(* PLC project booster_compressor, TwinForge TwinForge 0.1.0 *)
(* stored: creationDateTime 2026-07-23T22:04:36.214256+00:00 *)

PROGRAM MainProgram
  VAR
    TF_Cmp_MainProgram_R00_AnalogAlarms_0_1 : BOOL;  (* TwinForge comparison result for R00_AnalogAlarms rung 0 *)
    TF_Cmp_MainProgram_R00_AnalogAlarms_1_1 : BOOL;  (* TwinForge comparison result for R00_AnalogAlarms rung 1 *)
    TF_Cmp_MainProgram_R00_AnalogAlarms_2_1 : BOOL;  (* TwinForge comparison result for R00_AnalogAlarms rung 2 *)
    TF_Cmp_MainProgram_R00_AnalogAlarms_3_1 : BOOL;  (* TwinForge comparison result for R00_AnalogAlarms rung 3 *)
    TF_Cmp_MainProgram_R00_AnalogAlarms_4_1 : BOOL;  (* TwinForge comparison result for R00_AnalogAlarms rung 4 *)
    TF_Cmp_MainProgram_R00_AnalogAlarms_5_1 : BOOL;  (* TwinForge comparison result for R00_AnalogAlarms rung 5 *)
    TF_Cmp_MainProgram_R03_Trips_5_1 : BOOL;  (* TwinForge comparison result for R03_Trips rung 5 *)
    TF_Cmp_MainProgram_R03_Trips_7_1 : BOOL;  (* TwinForge comparison result for R03_Trips rung 7 *)
    TF_Cmp_MainProgram_R03_Trips_9_1 : BOOL;  (* TwinForge comparison result for R03_Trips rung 9 *)
    TF_Cmp_MainProgram_R03_Trips_10_1 : BOOL;  (* TwinForge comparison result for R03_Trips rung 10 *)
    TF_Cmp_MainProgram_R03_Trips_14_1 : BOOL;  (* TwinForge comparison result for R03_Trips rung 14 *)
    TF_Cmp_MainProgram_R03_Trips_15_1 : BOOL;  (* TwinForge comparison result for R03_Trips rung 15 *)
    TF_Cmp_MainProgram_R03_Trips_16_1 : BOOL;  (* TwinForge comparison result for R03_Trips rung 16 *)
    TF_Cmp_MainProgram_R03_Trips_17_1 : BOOL;  (* TwinForge comparison result for R03_Trips rung 17 *)
    TF_Cmp_MainProgram_R03_Trips_18_1 : BOOL;  (* TwinForge comparison result for R03_Trips rung 18 *)
    TF_Cmp_MainProgram_R03_Trips_19_1 : BOOL;  (* TwinForge comparison result for R03_Trips rung 19 *)
    TF_Cmp_MainProgram_R03_Trips_20_1 : BOOL;  (* TwinForge comparison result for R03_Trips rung 20 *)
    TF_Cmp_MainProgram_R03_Trips_21_1 : BOOL;  (* TwinForge comparison result for R03_Trips rung 21 *)
    TF_Cmp_MainProgram_R03_Trips_22_1 : BOOL;  (* TwinForge comparison result for R03_Trips rung 22 *)
    TF_Cmp_MainProgram_R04_Sequence_5_1 : BOOL;  (* TwinForge comparison result for R04_Sequence rung 5 *)
    TF_Cmp_MainProgram_R04_Sequence_5_2 : BOOL;  (* TwinForge comparison result for R04_Sequence rung 5 *)
    TF_Cmp_MainProgram_R04_Sequence_5_3 : BOOL;  (* TwinForge comparison result for R04_Sequence rung 5 *)
    TF_Cmp_MainProgram_R04_Sequence_6_1 : BOOL;  (* TwinForge comparison result for R04_Sequence rung 6 *)
    TF_Cmp_MainProgram_R04_Sequence_7_1 : BOOL;  (* TwinForge comparison result for R04_Sequence rung 7 *)
    TF_Cmp_MainProgram_R04_Sequence_8_1 : BOOL;  (* TwinForge comparison result for R04_Sequence rung 8 *)
    TF_Cmp_MainProgram_R04_Sequence_9_1 : BOOL;  (* TwinForge comparison result for R04_Sequence rung 9 *)
    TF_Cmp_MainProgram_R04_Sequence_9_2 : BOOL;  (* TwinForge comparison result for R04_Sequence rung 9 *)
    TF_Cmp_MainProgram_R04_Sequence_10_1 : BOOL;  (* TwinForge comparison result for R04_Sequence rung 10 *)
    TF_Cmp_MainProgram_R04_Sequence_10_2 : BOOL;  (* TwinForge comparison result for R04_Sequence rung 10 *)
    TF_Cmp_MainProgram_R04_Sequence_11_1 : BOOL;  (* TwinForge comparison result for R04_Sequence rung 11 *)
    TF_Cmp_MainProgram_R04_Sequence_11_2 : BOOL;  (* TwinForge comparison result for R04_Sequence rung 11 *)
    TF_Cmp_MainProgram_R04_Sequence_12_1 : BOOL;  (* TwinForge comparison result for R04_Sequence rung 12 *)
    TF_Cmp_MainProgram_R04_Sequence_13_1 : BOOL;  (* TwinForge comparison result for R04_Sequence rung 13 *)
    TF_Cmp_MainProgram_R04_Sequence_14_1 : BOOL;  (* TwinForge comparison result for R04_Sequence rung 14 *)
    TF_Cmp_MainProgram_R04_Sequence_15_1 : BOOL;  (* TwinForge comparison result for R04_Sequence rung 15 *)
    TF_Cmp_MainProgram_R04_Sequence_16_1 : BOOL;  (* TwinForge comparison result for R04_Sequence rung 16 *)
    TF_Cmp_MainProgram_R04_Sequence_17_1 : BOOL;  (* TwinForge comparison result for R04_Sequence rung 17 *)
    TF_Cmp_MainProgram_R04_Sequence_17_2 : BOOL;  (* TwinForge comparison result for R04_Sequence rung 17 *)
    TF_Cmp_MainProgram_R04_Sequence_18_1 : BOOL;  (* TwinForge comparison result for R04_Sequence rung 18 *)
    TF_Cmp_MainProgram_R04_Sequence_19_1 : BOOL;  (* TwinForge comparison result for R04_Sequence rung 19 *)
    TF_Cmp_MainProgram_R04_Sequence_20_1 : BOOL;  (* TwinForge comparison result for R04_Sequence rung 20 *)
    TF_Cmp_MainProgram_R04_Sequence_21_1 : BOOL;  (* TwinForge comparison result for R04_Sequence rung 21 *)
    TF_Cmp_MainProgram_R04_Sequence_22_1 : BOOL;  (* TwinForge comparison result for R04_Sequence rung 22 *)
    TF_Cmp_MainProgram_R04_Sequence_22_2 : BOOL;  (* TwinForge comparison result for R04_Sequence rung 22 *)
    TF_Cmp_MainProgram_R04_Sequence_23_1 : BOOL;  (* TwinForge comparison result for R04_Sequence rung 23 *)
    TF_Cmp_MainProgram_R04_Sequence_24_1 : BOOL;  (* TwinForge comparison result for R04_Sequence rung 24 *)
    TF_Cmp_MainProgram_R04_Sequence_25_1 : BOOL;  (* TwinForge comparison result for R04_Sequence rung 25 *)
    TF_Cmp_MainProgram_R04_Sequence_26_1 : BOOL;  (* TwinForge comparison result for R04_Sequence rung 26 *)
    TF_Cmp_MainProgram_R04_Sequence_26_2 : BOOL;  (* TwinForge comparison result for R04_Sequence rung 26 *)
    TF_Cmp_MainProgram_R04_Sequence_27_1 : BOOL;  (* TwinForge comparison result for R04_Sequence rung 27 *)
    TF_Cmp_MainProgram_R04_Sequence_28_1 : BOOL;  (* TwinForge comparison result for R04_Sequence rung 28 *)
    TF_Cmp_MainProgram_R04_Sequence_29_1 : BOOL;  (* TwinForge comparison result for R04_Sequence rung 29 *)
    TF_Cmp_MainProgram_R04_Sequence_30_1 : BOOL;  (* TwinForge comparison result for R04_Sequence rung 30 *)
    TF_Cmp_MainProgram_R04_Sequence_31_1 : BOOL;  (* TwinForge comparison result for R04_Sequence rung 31 *)
    TF_Cmp_MainProgram_R04_Sequence_32_1 : BOOL;  (* TwinForge comparison result for R04_Sequence rung 32 *)
    TF_Cmp_MainProgram_R04_Sequence_33_1 : BOOL;  (* TwinForge comparison result for R04_Sequence rung 33 *)
    TF_Cmp_MainProgram_R04_Sequence_33_2 : BOOL;  (* TwinForge comparison result for R04_Sequence rung 33 *)
    TF_Cmp_MainProgram_R04_Sequence_34_1 : BOOL;  (* TwinForge comparison result for R04_Sequence rung 34 *)
    TF_Cmp_MainProgram_R04_Sequence_34_2 : BOOL;  (* TwinForge comparison result for R04_Sequence rung 34 *)
    TF_Cmp_MainProgram_R04_Sequence_35_1 : BOOL;  (* TwinForge comparison result for R04_Sequence rung 35 *)
    TF_Cmp_MainProgram_R04_Sequence_36_1 : BOOL;  (* TwinForge comparison result for R04_Sequence rung 36 *)
    TF_Cmp_MainProgram_R04_Sequence_37_1 : BOOL;  (* TwinForge comparison result for R04_Sequence rung 37 *)
    TF_Cmp_MainProgram_R04_Sequence_37_2 : BOOL;  (* TwinForge comparison result for R04_Sequence rung 37 *)
    TF_Cmp_MainProgram_R04_Sequence_38_1 : BOOL;  (* TwinForge comparison result for R04_Sequence rung 38 *)
    TF_Cmp_MainProgram_R04_Sequence_39_1 : BOOL;  (* TwinForge comparison result for R04_Sequence rung 39 *)
    TF_Cmp_MainProgram_R04_Sequence_40_1 : BOOL;  (* TwinForge comparison result for R04_Sequence rung 40 *)
    TF_Cmp_MainProgram_R04_Sequence_41_1 : BOOL;  (* TwinForge comparison result for R04_Sequence rung 41 *)
    TF_Cmp_MainProgram_R04_Sequence_41_2 : BOOL;  (* TwinForge comparison result for R04_Sequence rung 41 *)
    TF_Cmp_MainProgram_R04_Sequence_42_1 : BOOL;  (* TwinForge comparison result for R04_Sequence rung 42 *)
    TF_Cmp_MainProgram_R04_Sequence_42_2 : BOOL;  (* TwinForge comparison result for R04_Sequence rung 42 *)
    TF_Cmp_MainProgram_R04_Sequence_43_1 : BOOL;  (* TwinForge comparison result for R04_Sequence rung 43 *)
    TF_Cmp_MainProgram_R04_Sequence_44_1 : BOOL;  (* TwinForge comparison result for R04_Sequence rung 44 *)
    TF_Cmp_MainProgram_R04_Sequence_45_1 : BOOL;  (* TwinForge comparison result for R04_Sequence rung 45 *)
    TF_Cmp_MainProgram_R04_Sequence_46_1 : BOOL;  (* TwinForge comparison result for R04_Sequence rung 46 *)
    TF_Cmp_MainProgram_R05_Devices_2_1 : BOOL;  (* TwinForge comparison result for R05_Devices rung 2 *)
    TF_Cmp_MainProgram_R05_Devices_4_1 : BOOL;  (* TwinForge comparison result for R05_Devices rung 4 *)
    TF_Cmp_MainProgram_R05_Devices_5_1 : BOOL;  (* TwinForge comparison result for R05_Devices rung 5 *)
    TF_Cmp_MainProgram_R05_Devices_6_1 : BOOL;  (* TwinForge comparison result for R05_Devices rung 6 *)
    TF_Cmp_MainProgram_R06_Control_5_1 : BOOL;  (* TwinForge comparison result for R06_Control rung 5 *)
    TF_Cmp_MainProgram_R06_Control_6_1 : BOOL;  (* TwinForge comparison result for R06_Control rung 6 *)
    TF_Cmp_MainProgram_R06_Control_7_1 : BOOL;  (* TwinForge comparison result for R06_Control rung 7 *)
    TF_Cmp_MainProgram_R06_Control_8_1 : BOOL;  (* TwinForge comparison result for R06_Control rung 8 *)
    TF_Cmp_MainProgram_R06_Control_10_1 : BOOL;  (* TwinForge comparison result for R06_Control rung 10 *)
    TF_Cmp_MainProgram_R06_Control_12_1 : BOOL;  (* TwinForge comparison result for R06_Control rung 12 *)
    TF_Cmp_MainProgram_R06_Control_14_1 : BOOL;  (* TwinForge comparison result for R06_Control rung 14 *)
    TF_Cmp_MainProgram_R06_Control_15_1 : BOOL;  (* TwinForge comparison result for R06_Control rung 15 *)
    TF_Cmp_MainProgram_R06_Control_16_1 : BOOL;  (* TwinForge comparison result for R06_Control rung 16 *)
    TF_Cmp_MainProgram_R06_Control_17_1 : BOOL;  (* TwinForge comparison result for R06_Control rung 17 *)
    TF_Cmp_MainProgram_R06_Control_18_1 : BOOL;  (* TwinForge comparison result for R06_Control rung 18 *)
    TF_Cmp_MainProgram_R06_Control_19_1 : BOOL;  (* TwinForge comparison result for R06_Control rung 19 *)
    TF_Cmp_MainProgram_R06_Control_20_1 : BOOL;  (* TwinForge comparison result for R06_Control rung 20 *)
    TF_Cmp_MainProgram_R06_Control_21_1 : BOOL;  (* TwinForge comparison result for R06_Control rung 21 *)
    TF_ONS_MainProgram_R03_Trips_24_FB : Standard.R_TRIG;  (* TwinForge rising-edge instance for Rockwell ONS storage operand TripActive *)
    TF_ONS_MainProgram_R03_Trips_24_IN : BOOL;  (* TwinForge ONS input for TripActive *)
    TF_ONS_MainProgram_R03_Trips_24_Pulse : BOOL;  (* TwinForge ONS one-scan pulse for TripActive *)
    TF_ONS_MainProgram_R03_Trips_24_Executed : BOOL;  (* TwinForge ONS execution for TripActive *)
  END_VAR
  VAR  (* added by the conversion: wires and edge detectors of the diagram *)
    _MOVE399_EN : BOOL;
    _MOVE449_EN : BOOL;
    _MOVE466_EN : BOOL;
    _MOVE478_EN : BOOL;
    _MOVE527_EN : BOOL;
    _MOVE553_EN : BOOL;
    _MOVE594_EN : BOOL;
    _MOVE611_EN : BOOL;
    _MOVE622_EN : BOOL;
    _MOVE674_EN : BOOL;
    _MOVE724_EN : BOOL;
    _MOVE889_EN : BOOL;
    _MOVE935_EN : BOOL;
    _MUL1037_EN : BOOL;
  END_VAR

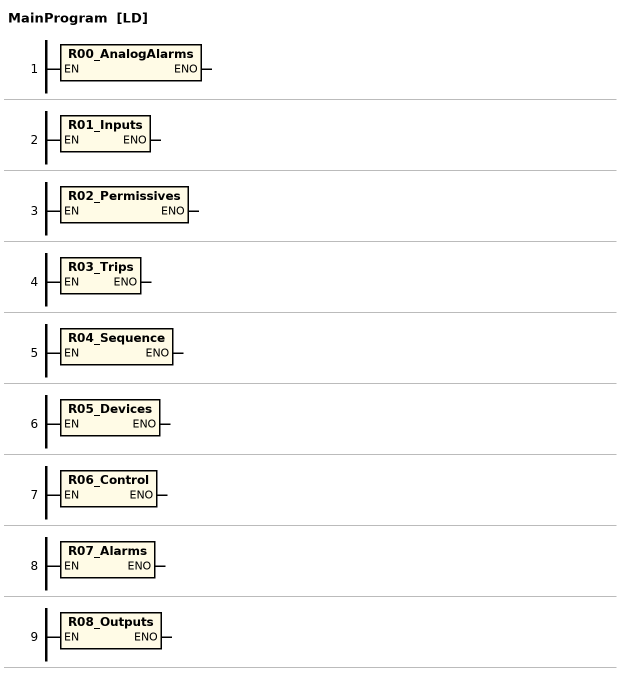
(* LD diagram, written out as Structured Text *)
(* ========================================================================
BOOSTER GAS COMPRESSOR STATION - PRODUCTION PROGRAM
Controller: 1756-L82E
I/O: Slot1=DI(16pt) Slot2=DI(16pt) Slot3=DO(16pt) Slot4=AI(4ch) Slot5=AO(8ch)
======================================================================== *)
R00_AnalogAlarms();
R01_Inputs();
R02_Permissives();
R03_Trips();
R04_Sequence();
R05_Devices();
R06_Control();
R07_Alarms();
R08_Outputs();

ACTION R00_AnalogAlarms:
(* LD diagram, written out as Structured Text *)
(* PT-102 Alarms *)
TF_Cmp_MainProgram_R00_AnalogAlarms_0_1 := PT102_PV > CFG_PT102_HH;
PT102_HH_Alm := TF_Cmp_MainProgram_R00_AnalogAlarms_0_1;
TF_Cmp_MainProgram_R00_AnalogAlarms_1_1 := PT102_PV > CFG_PT102_H;
PT102_H_Alm := TF_Cmp_MainProgram_R00_AnalogAlarms_1_1;
(* TT-102 Alarms *)
TF_Cmp_MainProgram_R00_AnalogAlarms_2_1 := TT102_PV > CFG_TT102_HH;
TT102_HH_Alm := TF_Cmp_MainProgram_R00_AnalogAlarms_2_1;
TF_Cmp_MainProgram_R00_AnalogAlarms_3_1 := TT102_PV > CFG_TT102_H;
TT102_H_Alm := TF_Cmp_MainProgram_R00_AnalogAlarms_3_1;
(* PT-201 Lube Oil Pressure Alarms *)
TF_Cmp_MainProgram_R00_AnalogAlarms_4_1 := PT201_PV < CFG_PT201_LL;
PT201_LL_Alm := TF_Cmp_MainProgram_R00_AnalogAlarms_4_1;
TF_Cmp_MainProgram_R00_AnalogAlarms_5_1 := PT201_PV < CFG_PT201_L;
PT201_L_Alm := TF_Cmp_MainProgram_R00_AnalogAlarms_5_1;
END_ACTION

ACTION R01_Inputs:
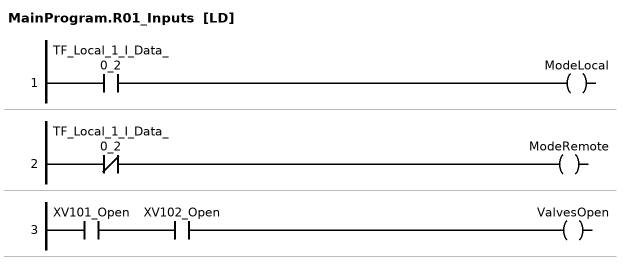
(* LD diagram, written out as Structured Text *)
(* Mode Selection *)
ModeLocal := TF_Local_1_I_Data_0_2;
ModeRemote := NOT TF_Local_1_I_Data_0_2;
(* Both Isolation Valves Open *)
ValvesOpen := XV101_Open AND XV102_Open;
END_ACTION

ACTION R02_Permissives:
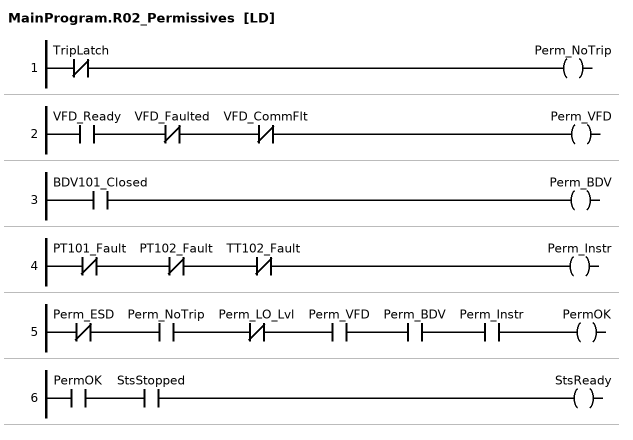
(* LD diagram, written out as Structured Text *)
(* No Active Trip Latched *)
Perm_NoTrip := NOT TripLatch;
(* VFD Ready and Not Faulted *)
Perm_VFD := VFD_Ready AND NOT VFD_Faulted AND NOT VFD_CommFlt;
(* Blowdown Valve Closed *)
Perm_BDV := BDV101_Closed;
(* Critical Instruments Healthy *)
Perm_Instr := NOT PT101_Fault AND NOT PT102_Fault AND NOT TT102_Fault;
(* Combine All Permissives *)
PermOK := NOT Perm_ESD AND Perm_NoTrip AND NOT Perm_LO_Lvl AND Perm_VFD AND Perm_BDV AND Perm_Instr;
(* Ready Status *)
StsReady := PermOK AND StsStopped;
END_ACTION

ACTION R03_Trips:
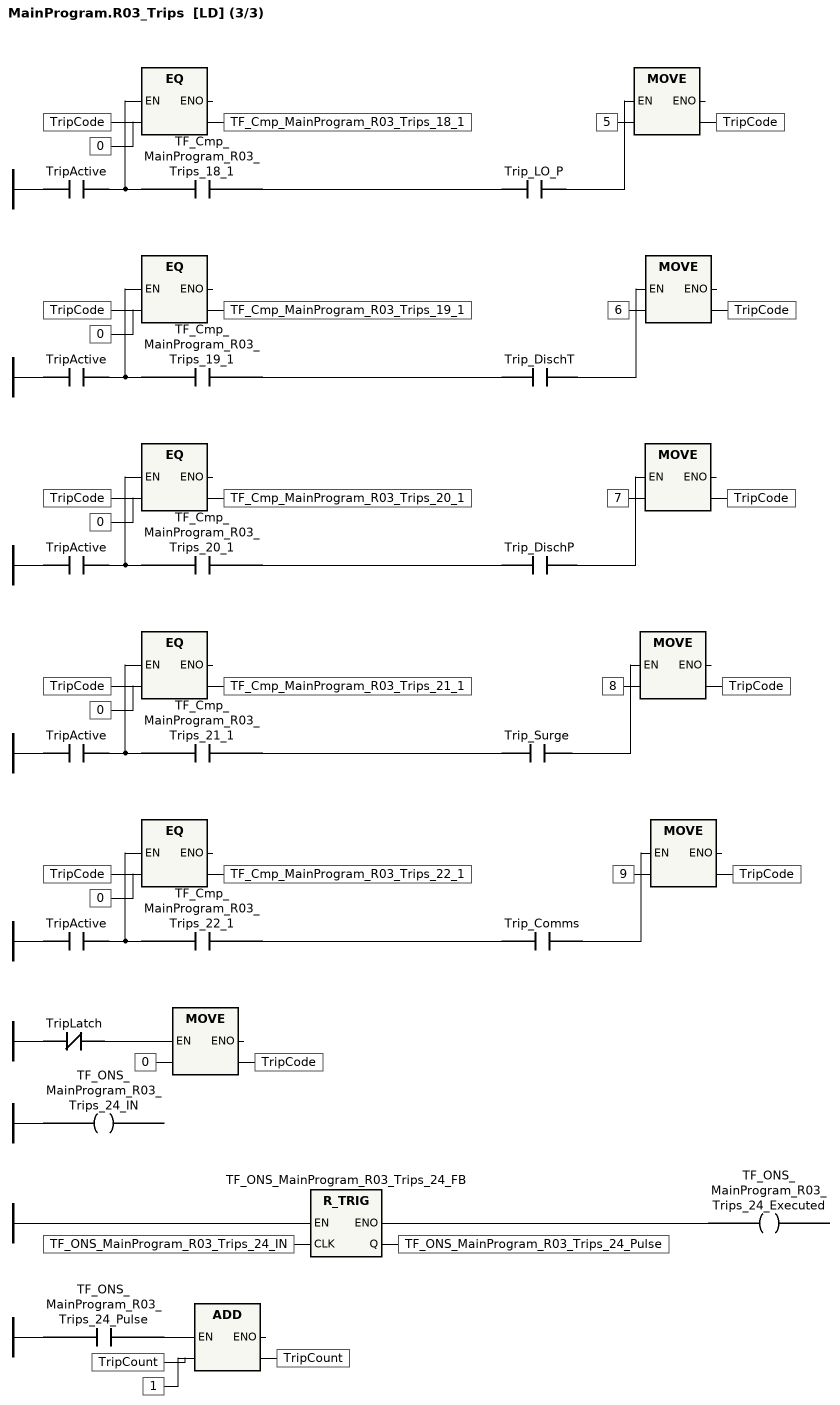
(* LD diagram, written out as Structured Text *)
(* ========== TRIP PROCESSING ========== *)
(* Fire Alarm *)
Trip_Fire := Alm_Fire;
(* VFD Fault while running *)
Trip_VFD := VFD_Faulted AND StsRunning;
(* VFD Comms Fault while running *)
Trip_Comms := VFD_CommFlt AND StsRunning;
(* ===== DELAYED TRIPS (2 sec filter) =====
Lube Oil Pressure Low-Low *)
TF_TMR_Trip_LO_IN := (Perm_LO_Lvl OR PT201_LL_Alm) AND StsRunning;
TMR_Trip_LO(IN := TF_TMR_Trip_LO_IN, PT := TIME#5000ms, Q => TF_TMR_Trip_LO_DN, ET => TF_TMR_Trip_LO_ET);
TF_TMR_Trip_LO_Executed := TMR_Trip_LO.ENO;
TF_Cmp_MainProgram_R03_Trips_5_1 := TF_TMR_Trip_LO_ET > DINT_TO_TIME(CFG_TripDelay);
Trip_LO_P := TF_Cmp_MainProgram_R03_Trips_5_1;
(* Discharge Temperature HH *)
TF_TMR_Trip_DischT_IN := TT102_HH_Alm AND StsRunning;
TMR_Trip_DischT(IN := TF_TMR_Trip_DischT_IN, PT := TIME#5000ms, Q => TF_TMR_Trip_DischT_DN, ET => TF_TMR_Trip_DischT_ET);
TF_TMR_Trip_DischT_Executed := TMR_Trip_DischT.ENO;
TF_Cmp_MainProgram_R03_Trips_7_1 := TF_TMR_Trip_DischT_ET > DINT_TO_TIME(CFG_TripDelay);
Trip_DischT := TF_Cmp_MainProgram_R03_Trips_7_1;
(* Discharge Pressure HH *)
TF_TMR_Trip_DischP_IN := PT102_HH_Alm AND StsRunning;
TMR_Trip_DischP(IN := TF_TMR_Trip_DischP_IN, PT := TIME#5000ms, Q => TF_TMR_Trip_DischP_DN, ET => TF_TMR_Trip_DischP_ET);
TF_TMR_Trip_DischP_Executed := TMR_Trip_DischP.ENO;
TF_Cmp_MainProgram_R03_Trips_9_1 := TF_TMR_Trip_DischP_ET > DINT_TO_TIME(CFG_TripDelay);
Trip_DischP := TF_Cmp_MainProgram_R03_Trips_9_1;
(* Surge Trip (low margin) *)
TF_Cmp_MainProgram_R03_Trips_10_1 := ASC_SurgeMargin < CFG_SurgeMarginTrip;
Trip_Surge := TF_Cmp_MainProgram_R03_Trips_10_1 AND StsRunning;
(* ===== COMBINE ALL TRIPS ===== *)
TripActive := NOT Trip_ESD OR Trip_Fire OR Trip_Vib OR Trip_VFD OR Trip_Comms OR Trip_LO_P OR Trip_DischT OR Trip_DischP OR Trip_Surge;
(* Latch Trip *)
IF TripActive THEN TripLatch := TRUE; END_IF;
(* Reset Trip (when condition cleared) *)
IF CmdReset AND NOT TripActive THEN TripLatch := FALSE; END_IF;
(* ===== FIRST-OUT TRIP CODE CAPTURE ===== *)
IF TripActive THEN TF_Cmp_MainProgram_R03_Trips_14_1 := TripCode = 0; END_IF;
IF TripActive AND TF_Cmp_MainProgram_R03_Trips_14_1 AND NOT Trip_ESD THEN TripCode := 1; END_IF;
IF TripActive THEN TF_Cmp_MainProgram_R03_Trips_15_1 := TripCode = 0; END_IF;
IF TripActive AND TF_Cmp_MainProgram_R03_Trips_15_1 AND Trip_Fire THEN TripCode := 2; END_IF;
IF TripActive THEN TF_Cmp_MainProgram_R03_Trips_16_1 := TripCode = 0; END_IF;
IF TripActive AND TF_Cmp_MainProgram_R03_Trips_16_1 AND Trip_Vib THEN TripCode := 3; END_IF;
IF TripActive THEN TF_Cmp_MainProgram_R03_Trips_17_1 := TripCode = 0; END_IF;
IF TripActive AND TF_Cmp_MainProgram_R03_Trips_17_1 AND Trip_VFD THEN TripCode := 4; END_IF;
IF TripActive THEN TF_Cmp_MainProgram_R03_Trips_18_1 := TripCode = 0; END_IF;
IF TripActive AND TF_Cmp_MainProgram_R03_Trips_18_1 AND Trip_LO_P THEN TripCode := 5; END_IF;
IF TripActive THEN TF_Cmp_MainProgram_R03_Trips_19_1 := TripCode = 0; END_IF;
IF TripActive AND TF_Cmp_MainProgram_R03_Trips_19_1 AND Trip_DischT THEN TripCode := 6; END_IF;
IF TripActive THEN TF_Cmp_MainProgram_R03_Trips_20_1 := TripCode = 0; END_IF;
IF TripActive AND TF_Cmp_MainProgram_R03_Trips_20_1 AND Trip_DischP THEN TripCode := 7; END_IF;
IF TripActive THEN TF_Cmp_MainProgram_R03_Trips_21_1 := TripCode = 0; END_IF;
IF TripActive AND TF_Cmp_MainProgram_R03_Trips_21_1 AND Trip_Surge THEN TripCode := 8; END_IF;
IF TripActive THEN TF_Cmp_MainProgram_R03_Trips_22_1 := TripCode = 0; END_IF;
IF TripActive AND TF_Cmp_MainProgram_R03_Trips_22_1 AND Trip_Comms THEN TripCode := 9; END_IF;
(* Clear trip code when reset *)
IF NOT TripLatch THEN TripCode := 0; END_IF;
(* Trip Counter *)
TF_ONS_MainProgram_R03_Trips_24_IN := TRUE;
TF_ONS_MainProgram_R03_Trips_24_FB(CLK := TF_ONS_MainProgram_R03_Trips_24_IN, Q => TF_ONS_MainProgram_R03_Trips_24_Pulse);
TF_ONS_MainProgram_R03_Trips_24_Executed := TF_ONS_MainProgram_R03_Trips_24_FB.ENO;
IF TF_ONS_MainProgram_R03_Trips_24_Pulse THEN TripCount := TripCount + 1; END_IF;
END_ACTION

ACTION R04_Sequence:
(* LD diagram, written out as Structured Text *)
(* ========== SEQUENCE STATE MACHINE ==========
State: 0=Stopped 10=Prelube 20=OpenValves 30=StartVFD 40=Warmup 50=Running 60=Shutdown 90=Tripped 95=ESD *)
(* ===== COMMAND PROCESSING =====
Start Command from Local PB or HMI *)
IF (TF_Local_1_I_Data_1 AND ModeLocal OR HMI_Start AND ModeRemote) AND NOT ONS_Start THEN CmdStart := TRUE; END_IF;
ONS_Start := (TF_Local_1_I_Data_1 AND ModeLocal OR HMI_Start AND ModeRemote) AND NOT ONS_Start;
(* Stop Command (Local PB always works) *)
IF TF_Local_1_I_Data_2 OR HMI_Stop THEN CmdStop := TRUE; END_IF;
(* Reset Command *)
IF (TF_Local_1_I_Data_3 AND ModeLocal OR HMI_Reset AND ModeRemote) AND NOT ONS_Reset THEN CmdReset := TRUE; END_IF;
ONS_Reset := (TF_Local_1_I_Data_3 AND ModeLocal OR HMI_Reset AND ModeRemote) AND NOT ONS_Reset;
(* ===== ESD/FIRE - HIGHEST PRIORITY ===== *)
IF NOT Trip_ESD OR Trip_Fire THEN State := 95; END_IF;
(* ===== TRIP PRIORITY ===== *)
IF TripActive THEN TF_Cmp_MainProgram_R04_Sequence_5_1 := State <> 0; END_IF;
IF TripActive AND TF_Cmp_MainProgram_R04_Sequence_5_1 THEN TF_Cmp_MainProgram_R04_Sequence_5_2 := State <> 90; END_IF;
IF TripActive AND TF_Cmp_MainProgram_R04_Sequence_5_1 AND TF_Cmp_MainProgram_R04_Sequence_5_2 THEN TF_Cmp_MainProgram_R04_Sequence_5_3 := State <> 95; END_IF;
IF TripActive AND TF_Cmp_MainProgram_R04_Sequence_5_1 AND TF_Cmp_MainProgram_R04_Sequence_5_2 AND TF_Cmp_MainProgram_R04_Sequence_5_3 THEN State := 90; END_IF;
(* ===== STATE 0: STOPPED ===== *)
TF_Cmp_MainProgram_R04_Sequence_6_1 := State = 0;
StsStopped := TF_Cmp_MainProgram_R04_Sequence_6_1;
IF TF_Cmp_MainProgram_R04_Sequence_6_1 THEN StsStarting := FALSE; END_IF;
IF TF_Cmp_MainProgram_R04_Sequence_6_1 THEN StsRunning := FALSE; END_IF;
IF TF_Cmp_MainProgram_R04_Sequence_6_1 THEN StsStopping := FALSE; END_IF;
IF TF_Cmp_MainProgram_R04_Sequence_6_1 THEN StsTripped := FALSE; END_IF;
IF TF_Cmp_MainProgram_R04_Sequence_6_1 THEN StsESD := FALSE; END_IF;
IF TF_Cmp_MainProgram_R04_Sequence_6_1 THEN VFD_CmdStart := FALSE; END_IF;
IF TF_Cmp_MainProgram_R04_Sequence_6_1 THEN LO_PumpCmd := FALSE; END_IF;
IF TF_Cmp_MainProgram_R04_Sequence_6_1 THEN LO_PressOK := FALSE; END_IF;
(* Transition: STOPPED -> PRELUBE on Start *)
TF_Cmp_MainProgram_R04_Sequence_7_1 := State = 0;
_MOVE399_EN := TF_Cmp_MainProgram_R04_Sequence_7_1 AND CmdStart AND PermOK;
IF _MOVE399_EN THEN State := 10; END_IF;
IF _MOVE399_EN THEN StartCount := StartCount + 1; END_IF;
TMR_Prelube(EN := _MOVE399_EN, IN := FALSE, PT := TIME#100000ms, Q => TF_TMR_Prelube_DN, ET => TF_TMR_Prelube_ET);
IF TMR_Prelube.ENO THEN CmdStart := FALSE; END_IF;
(* ===== STATE 10: PRELUBE ===== *)
TF_Cmp_MainProgram_R04_Sequence_8_1 := State = 10;
IF TF_Cmp_MainProgram_R04_Sequence_8_1 THEN StsStopped := FALSE; END_IF;
StsStarting := TF_Cmp_MainProgram_R04_Sequence_8_1;
LO_PumpCmd := TF_Cmp_MainProgram_R04_Sequence_8_1;
TF_TMR_Prelube_IN := TF_Cmp_MainProgram_R04_Sequence_8_1;
TMR_Prelube(IN := TF_TMR_Prelube_IN, PT := TIME#100000ms, Q => TF_TMR_Prelube_DN, ET => TF_TMR_Prelube_ET);
TF_TMR_Prelube_Executed := TMR_Prelube.ENO;
(* Check Lube Oil Pressure OK *)
TF_Cmp_MainProgram_R04_Sequence_9_1 := State = 10;
IF TF_Cmp_MainProgram_R04_Sequence_9_1 THEN TF_Cmp_MainProgram_R04_Sequence_9_2 := PT201_PV >= CFG_LO_Press_Min; END_IF;
LO_PressOK := TF_Cmp_MainProgram_R04_Sequence_9_1 AND TF_Cmp_MainProgram_R04_Sequence_9_2;
(* Transition: PRELUBE -> OPEN_VALVES *)
TF_Cmp_MainProgram_R04_Sequence_10_1 := State = 10;
IF TF_Cmp_MainProgram_R04_Sequence_10_1 AND LO_PressOK THEN TF_Cmp_MainProgram_R04_Sequence_10_2 := TF_TMR_Prelube_ET > DINT_TO_TIME(CFG_PrelubeTime); END_IF;
_MOVE449_EN := TF_Cmp_MainProgram_R04_Sequence_10_1 AND LO_PressOK AND TF_Cmp_MainProgram_R04_Sequence_10_2;
IF _MOVE449_EN THEN State := 20; END_IF;
TMR_Valve(EN := _MOVE449_EN, IN := FALSE, PT := TIME#100000ms, Q => TF_TMR_Valve_DN, ET => TF_TMR_Valve_ET);
(* Timeout: PRELUBE -> TRIPPED (failed to build pressure) *)
TF_Cmp_MainProgram_R04_Sequence_11_1 := State = 10;
IF TF_Cmp_MainProgram_R04_Sequence_11_1 THEN TF_Cmp_MainProgram_R04_Sequence_11_2 := TF_TMR_Prelube_ET > DINT_TO_TIME(CFG_PrelubeTimeout); END_IF;
IF TF_Cmp_MainProgram_R04_Sequence_11_1 AND TF_Cmp_MainProgram_R04_Sequence_11_2 THEN TripLatch := TRUE; END_IF;
_MOVE466_EN := TF_Cmp_MainProgram_R04_Sequence_11_1 AND TF_Cmp_MainProgram_R04_Sequence_11_2;
IF _MOVE466_EN THEN TripCode := 5; END_IF;
IF _MOVE466_EN THEN State := 90; END_IF;
(* Abort: PRELUBE -> SHUTDOWN on Stop *)
TF_Cmp_MainProgram_R04_Sequence_12_1 := State = 10;
_MOVE478_EN := TF_Cmp_MainProgram_R04_Sequence_12_1 AND CmdStop;
IF _MOVE478_EN THEN State := 60; END_IF;
TMR_PostLube(EN := _MOVE478_EN, IN := FALSE, PT := TIME#400000ms, Q => TF_TMR_PostLube_DN, ET => TF_TMR_PostLube_ET);
IF TMR_PostLube.ENO THEN CmdStop := FALSE; END_IF;
(* ===== STATE 20: OPEN VALVES ===== *)
TF_Cmp_MainProgram_R04_Sequence_13_1 := State = 20;
StsStarting := TF_Cmp_MainProgram_R04_Sequence_13_1;
LO_PumpCmd := TF_Cmp_MainProgram_R04_Sequence_13_1;
XV101_CmdOpen := TF_Cmp_MainProgram_R04_Sequence_13_1;
IF TF_Cmp_MainProgram_R04_Sequence_13_1 THEN XV101_CmdClose := FALSE; END_IF;
IF TF_Cmp_MainProgram_R04_Sequence_13_1 THEN BDV101_CmdOpen := FALSE; END_IF;
TF_Cmp_MainProgram_R04_Sequence_14_1 := State = 20;
TF_TMR_Valve_IN := TF_Cmp_MainProgram_R04_Sequence_14_1;
TMR_Valve(IN := TF_TMR_Valve_IN, PT := TIME#100000ms, Q => TF_TMR_Valve_DN, ET => TF_TMR_Valve_ET);
TF_TMR_Valve_Executed := TMR_Valve.ENO;
(* Open discharge valve after suction opens *)
TF_Cmp_MainProgram_R04_Sequence_15_1 := State = 20;
XV102_CmdOpen := TF_Cmp_MainProgram_R04_Sequence_15_1 AND XV101_Open;
IF TF_Cmp_MainProgram_R04_Sequence_15_1 AND XV101_Open THEN XV102_CmdClose := FALSE; END_IF;
(* Transition: OPEN_VALVES -> START_VFD *)
TF_Cmp_MainProgram_R04_Sequence_16_1 := State = 20;
_MOVE527_EN := TF_Cmp_MainProgram_R04_Sequence_16_1 AND ValvesOpen;
IF _MOVE527_EN THEN State := 30; END_IF;
TMR_VFDStart(EN := _MOVE527_EN, IN := FALSE, PT := TIME#60000ms, Q => TF_TMR_VFDStart_DN, ET => TF_TMR_VFDStart_ET);
(* Timeout: OPEN_VALVES -> TRIPPED *)
TF_Cmp_MainProgram_R04_Sequence_17_1 := State = 20;
IF TF_Cmp_MainProgram_R04_Sequence_17_1 THEN TF_Cmp_MainProgram_R04_Sequence_17_2 := TF_TMR_Valve_ET > DINT_TO_TIME(CFG_ValveTimeout); END_IF;
IF TF_Cmp_MainProgram_R04_Sequence_17_1 AND TF_Cmp_MainProgram_R04_Sequence_17_2 THEN TripLatch := TRUE; END_IF;
IF TF_Cmp_MainProgram_R04_Sequence_17_1 AND TF_Cmp_MainProgram_R04_Sequence_17_2 THEN State := 90; END_IF;
TF_Cmp_MainProgram_R04_Sequence_18_1 := State = 20;
_MOVE553_EN := TF_Cmp_MainProgram_R04_Sequence_18_1 AND CmdStop;
IF _MOVE553_EN THEN State := 60; END_IF;
TMR_PostLube(EN := _MOVE553_EN, IN := FALSE, PT := TIME#400000ms, Q => TF_TMR_PostLube_DN, ET => TF_TMR_PostLube_ET);
IF TMR_PostLube.ENO THEN CmdStop := FALSE; END_IF;
(* ===== STATE 30: START VFD ===== *)
TF_Cmp_MainProgram_R04_Sequence_19_1 := State = 30;
StsStarting := TF_Cmp_MainProgram_R04_Sequence_19_1;
LO_PumpCmd := TF_Cmp_MainProgram_R04_Sequence_19_1;
XV101_CmdOpen := TF_Cmp_MainProgram_R04_Sequence_19_1;
XV102_CmdOpen := TF_Cmp_MainProgram_R04_Sequence_19_1;
VFD_CmdStart := TF_Cmp_MainProgram_R04_Sequence_19_1;
IF TF_Cmp_MainProgram_R04_Sequence_19_1 THEN TF_Local_5_O_Ch1Data_8 := CFG_SpeedStart; END_IF;
TF_Cmp_MainProgram_R04_Sequence_20_1 := State = 30;
TF_TMR_VFDStart_IN := TF_Cmp_MainProgram_R04_Sequence_20_1;
TMR_VFDStart(IN := TF_TMR_VFDStart_IN, PT := TIME#60000ms, Q => TF_TMR_VFDStart_DN, ET => TF_TMR_VFDStart_ET);
TF_TMR_VFDStart_Executed := TMR_VFDStart.ENO;
(* Transition: START_VFD -> WARMUP *)
TF_Cmp_MainProgram_R04_Sequence_21_1 := State = 30;
_MOVE594_EN := TF_Cmp_MainProgram_R04_Sequence_21_1 AND VFD_Running;
IF _MOVE594_EN THEN State := 40; END_IF;
TMR_Warmup(EN := _MOVE594_EN, IN := FALSE, PT := TIME#100000ms, Q => TF_TMR_Warmup_DN, ET => TF_TMR_Warmup_ET);
(* Timeout: START_VFD -> TRIPPED *)
TF_Cmp_MainProgram_R04_Sequence_22_1 := State = 30;
IF TF_Cmp_MainProgram_R04_Sequence_22_1 THEN TF_Cmp_MainProgram_R04_Sequence_22_2 := TF_TMR_VFDStart_ET > DINT_TO_TIME(CFG_VFDStartTimeout); END_IF;
IF TF_Cmp_MainProgram_R04_Sequence_22_1 AND TF_Cmp_MainProgram_R04_Sequence_22_2 THEN TripLatch := TRUE; END_IF;
_MOVE611_EN := TF_Cmp_MainProgram_R04_Sequence_22_1 AND TF_Cmp_MainProgram_R04_Sequence_22_2;
IF _MOVE611_EN THEN TripCode := 4; END_IF;
IF _MOVE611_EN THEN State := 90; END_IF;
TF_Cmp_MainProgram_R04_Sequence_23_1 := State = 30;
_MOVE622_EN := TF_Cmp_MainProgram_R04_Sequence_23_1 AND CmdStop;
IF _MOVE622_EN THEN State := 60; END_IF;
TMR_PostLube(EN := _MOVE622_EN, IN := FALSE, PT := TIME#400000ms, Q => TF_TMR_PostLube_DN, ET => TF_TMR_PostLube_ET);
IF TMR_PostLube.ENO THEN CmdStop := FALSE; END_IF;
(* ===== STATE 40: WARMUP ===== *)
TF_Cmp_MainProgram_R04_Sequence_24_1 := State = 40;
StsStarting := TF_Cmp_MainProgram_R04_Sequence_24_1;
LO_PumpCmd := TF_Cmp_MainProgram_R04_Sequence_24_1;
XV101_CmdOpen := TF_Cmp_MainProgram_R04_Sequence_24_1;
XV102_CmdOpen := TF_Cmp_MainProgram_R04_Sequence_24_1;
VFD_CmdStart := TF_Cmp_MainProgram_R04_Sequence_24_1;
ASC_Enable := TF_Cmp_MainProgram_R04_Sequence_24_1;
TF_Cmp_MainProgram_R04_Sequence_25_1 := State = 40;
TF_TMR_Warmup_IN := TF_Cmp_MainProgram_R04_Sequence_25_1;
TMR_Warmup(IN := TF_TMR_Warmup_IN, PT := TIME#100000ms, Q => TF_TMR_Warmup_DN, ET => TF_TMR_Warmup_ET);
TF_TMR_Warmup_Executed := TMR_Warmup.ENO;
(* Transition: WARMUP -> RUNNING *)
TF_Cmp_MainProgram_R04_Sequence_26_1 := State = 40;
IF TF_Cmp_MainProgram_R04_Sequence_26_1 THEN TF_Cmp_MainProgram_R04_Sequence_26_2 := TF_TMR_Warmup_ET > DINT_TO_TIME(CFG_WarmupTime); END_IF;
IF TF_Cmp_MainProgram_R04_Sequence_26_1 AND TF_Cmp_MainProgram_R04_Sequence_26_2 THEN State := 50; END_IF;
TF_Cmp_MainProgram_R04_Sequence_27_1 := State = 40;
_MOVE674_EN := TF_Cmp_MainProgram_R04_Sequence_27_1 AND CmdStop;
IF _MOVE674_EN THEN State := 60; END_IF;
TMR_PostLube(EN := _MOVE674_EN, IN := FALSE, PT := TIME#400000ms, Q => TF_TMR_PostLube_DN, ET => TF_TMR_PostLube_ET);
IF TMR_PostLube.ENO THEN CmdStop := FALSE; END_IF;
(* ===== STATE 50: RUNNING ===== *)
TF_Cmp_MainProgram_R04_Sequence_28_1 := State = 50;
IF TF_Cmp_MainProgram_R04_Sequence_28_1 THEN StsStarting := FALSE; END_IF;
StsRunning := TF_Cmp_MainProgram_R04_Sequence_28_1;
LO_PumpCmd := TF_Cmp_MainProgram_R04_Sequence_28_1;
VFD_CmdStart := TF_Cmp_MainProgram_R04_Sequence_28_1;
XV101_CmdOpen := TF_Cmp_MainProgram_R04_Sequence_28_1;
XV102_CmdOpen := TF_Cmp_MainProgram_R04_Sequence_28_1;
PID_Enable := TF_Cmp_MainProgram_R04_Sequence_28_1;
PID_Auto := TF_Cmp_MainProgram_R04_Sequence_28_1;
ASC_Enable := TF_Cmp_MainProgram_R04_Sequence_28_1;
ASC_Auto := TF_Cmp_MainProgram_R04_Sequence_28_1;
(* Speed from PID output *)
TF_Cmp_MainProgram_R04_Sequence_29_1 := State = 50;
IF TF_Cmp_MainProgram_R04_Sequence_29_1 THEN TF_Local_5_O_Ch1Data_8 := PID_Out; END_IF;
(* Run Hours Accumulation *)
TF_Cmp_MainProgram_R04_Sequence_30_1 := State = 50;
IF TF_Cmp_MainProgram_R04_Sequence_30_1 THEN RunHours := RunHours + 0.0000278; END_IF;
(* Transition: RUNNING -> SHUTDOWN on Stop *)
TF_Cmp_MainProgram_R04_Sequence_31_1 := State = 50;
_MOVE724_EN := TF_Cmp_MainProgram_R04_Sequence_31_1 AND CmdStop;
IF _MOVE724_EN THEN State := 60; END_IF;
TMR_PostLube(EN := _MOVE724_EN, IN := FALSE, PT := TIME#400000ms, Q => TF_TMR_PostLube_DN, ET => TF_TMR_PostLube_ET);
IF TMR_PostLube.ENO THEN CmdStop := FALSE; END_IF;
(* ===== STATE 60: NORMAL SHUTDOWN ===== *)
TF_Cmp_MainProgram_R04_Sequence_32_1 := State = 60;
IF TF_Cmp_MainProgram_R04_Sequence_32_1 THEN StsRunning := FALSE; END_IF;
StsStopping := TF_Cmp_MainProgram_R04_Sequence_32_1;
IF TF_Cmp_MainProgram_R04_Sequence_32_1 THEN PID_Enable := FALSE; END_IF;
IF TF_Cmp_MainProgram_R04_Sequence_32_1 THEN TF_Local_5_O_Ch0Data_4 := CFG_RecycleShutdown; END_IF;
LO_PumpCmd := TF_Cmp_MainProgram_R04_Sequence_32_1;
(* Ramp Down VFD Speed *)
TF_Cmp_MainProgram_R04_Sequence_33_1 := State = 60;
IF TF_Cmp_MainProgram_R04_Sequence_33_1 THEN TF_Cmp_MainProgram_R04_Sequence_33_2 := TF_Local_5_O_Ch1Data_8 > CFG_SpeedMin; END_IF;
IF TF_Cmp_MainProgram_R04_Sequence_33_1 AND TF_Cmp_MainProgram_R04_Sequence_33_2 THEN TF_Local_5_O_Ch1Data_8 := TF_Local_5_O_Ch1Data_8 - 1.0; END_IF;
(* Stop VFD at Minimum Speed *)
TF_Cmp_MainProgram_R04_Sequence_34_1 := State = 60;
IF TF_Cmp_MainProgram_R04_Sequence_34_1 THEN TF_Cmp_MainProgram_R04_Sequence_34_2 := TF_Local_5_O_Ch1Data_8 <= CFG_SpeedMin; END_IF;
IF TF_Cmp_MainProgram_R04_Sequence_34_1 AND TF_Cmp_MainProgram_R04_Sequence_34_2 THEN VFD_CmdStart := FALSE; END_IF;
VFD_CmdStop := TF_Cmp_MainProgram_R04_Sequence_34_1 AND TF_Cmp_MainProgram_R04_Sequence_34_2;
(* After VFD stops: Open blowdown, close isolation *)
TF_Cmp_MainProgram_R04_Sequence_35_1 := State = 60;
BDV101_CmdOpen := TF_Cmp_MainProgram_R04_Sequence_35_1 AND NOT VFD_Running;
IF TF_Cmp_MainProgram_R04_Sequence_35_1 AND NOT VFD_Running THEN XV102_CmdOpen := FALSE; END_IF;
XV102_CmdClose := TF_Cmp_MainProgram_R04_Sequence_35_1 AND NOT VFD_Running;
IF TF_Cmp_MainProgram_R04_Sequence_35_1 AND NOT VFD_Running THEN XV101_CmdOpen := FALSE; END_IF;
XV101_CmdClose := TF_Cmp_MainProgram_R04_Sequence_35_1 AND NOT VFD_Running;
(* Post-Lube Timer *)
TF_Cmp_MainProgram_R04_Sequence_36_1 := State = 60;
TF_TMR_PostLube_IN := TF_Cmp_MainProgram_R04_Sequence_36_1 AND NOT VFD_Running;
TMR_PostLube(IN := TF_TMR_PostLube_IN, PT := TIME#400000ms, Q => TF_TMR_PostLube_DN, ET => TF_TMR_PostLube_ET);
TF_TMR_PostLube_Executed := TMR_PostLube.ENO;
(* Transition: SHUTDOWN -> STOPPED *)
TF_Cmp_MainProgram_R04_Sequence_37_1 := State = 60;
IF TF_Cmp_MainProgram_R04_Sequence_37_1 AND NOT VFD_Running THEN TF_Cmp_MainProgram_R04_Sequence_37_2 := TF_TMR_PostLube_ET > DINT_TO_TIME(CFG_PostLubeTime); END_IF;
IF TF_Cmp_MainProgram_R04_Sequence_37_1 AND NOT VFD_Running AND TF_Cmp_MainProgram_R04_Sequence_37_2 THEN LO_PumpCmd := FALSE; END_IF;
IF TF_Cmp_MainProgram_R04_Sequence_37_1 AND NOT VFD_Running AND TF_Cmp_MainProgram_R04_Sequence_37_2 THEN State := 0; END_IF;
(* ===== STATE 90: TRIPPED ===== *)
TF_Cmp_MainProgram_R04_Sequence_38_1 := State = 90;
IF TF_Cmp_MainProgram_R04_Sequence_38_1 THEN StsRunning := FALSE; END_IF;
IF TF_Cmp_MainProgram_R04_Sequence_38_1 THEN StsStarting := FALSE; END_IF;
IF TF_Cmp_MainProgram_R04_Sequence_38_1 THEN StsStopping := FALSE; END_IF;
StsTripped := TF_Cmp_MainProgram_R04_Sequence_38_1;
IF TF_Cmp_MainProgram_R04_Sequence_38_1 THEN TF_Local_5_O_Ch0Data_4 := 100.0; END_IF;
IF TF_Cmp_MainProgram_R04_Sequence_38_1 THEN VFD_CmdStart := FALSE; END_IF;
VFD_CmdStop := TF_Cmp_MainProgram_R04_Sequence_38_1;
IF TF_Cmp_MainProgram_R04_Sequence_38_1 THEN TF_Local_5_O_Ch1Data_8 := 0.0; END_IF;
TF_Cmp_MainProgram_R04_Sequence_39_1 := State = 90;
BDV101_CmdOpen := TF_Cmp_MainProgram_R04_Sequence_39_1;
IF TF_Cmp_MainProgram_R04_Sequence_39_1 THEN XV101_CmdOpen := FALSE; END_IF;
XV101_CmdClose := TF_Cmp_MainProgram_R04_Sequence_39_1;
IF TF_Cmp_MainProgram_R04_Sequence_39_1 THEN XV102_CmdOpen := FALSE; END_IF;
XV102_CmdClose := TF_Cmp_MainProgram_R04_Sequence_39_1;
IF TF_Cmp_MainProgram_R04_Sequence_39_1 THEN PID_Enable := FALSE; END_IF;
IF TF_Cmp_MainProgram_R04_Sequence_39_1 THEN ASC_Enable := FALSE; END_IF;
(* Extended Post-Lube After Trip *)
TF_Cmp_MainProgram_R04_Sequence_40_1 := State = 90;
TF_TMR_PostLube_IN := TF_Cmp_MainProgram_R04_Sequence_40_1;
TMR_PostLube(IN := TF_TMR_PostLube_IN, PT := TIME#400000ms, Q => TF_TMR_PostLube_DN, ET => TF_TMR_PostLube_ET);
TF_TMR_PostLube_Executed := TMR_PostLube.ENO;
TF_Cmp_MainProgram_R04_Sequence_41_1 := State = 90;
IF TF_Cmp_MainProgram_R04_Sequence_41_1 THEN TF_Cmp_MainProgram_R04_Sequence_41_2 := TF_TMR_PostLube_ET < DINT_TO_TIME(CFG_PostLubeTripTime); END_IF;
LO_PumpCmd := TF_Cmp_MainProgram_R04_Sequence_41_1 AND TF_Cmp_MainProgram_R04_Sequence_41_2;
TF_Cmp_MainProgram_R04_Sequence_42_1 := State = 90;
IF TF_Cmp_MainProgram_R04_Sequence_42_1 THEN TF_Cmp_MainProgram_R04_Sequence_42_2 := TF_TMR_PostLube_ET >= DINT_TO_TIME(CFG_PostLubeTripTime); END_IF;
IF TF_Cmp_MainProgram_R04_Sequence_42_1 AND TF_Cmp_MainProgram_R04_Sequence_42_2 THEN LO_PumpCmd := FALSE; END_IF;
(* Transition: TRIPPED -> STOPPED on Reset *)
TF_Cmp_MainProgram_R04_Sequence_43_1 := State = 90;
IF TF_Cmp_MainProgram_R04_Sequence_43_1 AND CmdReset AND NOT TripActive THEN TripLatch := FALSE; END_IF;
_MOVE889_EN := TF_Cmp_MainProgram_R04_Sequence_43_1 AND CmdReset AND NOT TripActive;
IF _MOVE889_EN THEN TripCode := 0; END_IF;
IF _MOVE889_EN THEN State := 0; END_IF;
IF _MOVE889_EN THEN CmdReset := FALSE; END_IF;
(* ===== STATE 95: ESD ACTIVE ===== *)
TF_Cmp_MainProgram_R04_Sequence_44_1 := State = 95;
IF TF_Cmp_MainProgram_R04_Sequence_44_1 THEN StsRunning := FALSE; END_IF;
IF TF_Cmp_MainProgram_R04_Sequence_44_1 THEN StsStarting := FALSE; END_IF;
StsTripped := TF_Cmp_MainProgram_R04_Sequence_44_1;
StsESD := TF_Cmp_MainProgram_R04_Sequence_44_1;
IF TF_Cmp_MainProgram_R04_Sequence_44_1 THEN VFD_CmdStart := FALSE; END_IF;
VFD_CmdStop := TF_Cmp_MainProgram_R04_Sequence_44_1;
IF TF_Cmp_MainProgram_R04_Sequence_44_1 THEN TF_Local_5_O_Ch1Data_8 := 0.0; END_IF;
IF TF_Cmp_MainProgram_R04_Sequence_44_1 THEN LO_PumpCmd := FALSE; END_IF;
IF TF_Cmp_MainProgram_R04_Sequence_44_1 THEN FanCmd := FALSE; END_IF;
TF_Cmp_MainProgram_R04_Sequence_45_1 := State = 95;
IF TF_Cmp_MainProgram_R04_Sequence_45_1 THEN XV101_CmdOpen := FALSE; END_IF;
XV101_CmdClose := TF_Cmp_MainProgram_R04_Sequence_45_1;
IF TF_Cmp_MainProgram_R04_Sequence_45_1 THEN XV102_CmdOpen := FALSE; END_IF;
XV102_CmdClose := TF_Cmp_MainProgram_R04_Sequence_45_1;
BDV101_CmdOpen := TF_Cmp_MainProgram_R04_Sequence_45_1;
IF TF_Cmp_MainProgram_R04_Sequence_45_1 THEN TF_Local_5_O_Ch0Data_4 := 100.0; END_IF;
IF TF_Cmp_MainProgram_R04_Sequence_45_1 THEN PID_Enable := FALSE; END_IF;
IF TF_Cmp_MainProgram_R04_Sequence_45_1 THEN ASC_Enable := FALSE; END_IF;
(* Transition: ESD -> TRIPPED when ESD restored *)
TF_Cmp_MainProgram_R04_Sequence_46_1 := State = 95;
_MOVE935_EN := TF_Cmp_MainProgram_R04_Sequence_46_1 AND Trip_ESD AND NOT Trip_Fire;
IF _MOVE935_EN THEN State := 90; END_IF;
TMR_PostLube(EN := _MOVE935_EN, IN := FALSE, PT := TIME#400000ms, Q => TF_TMR_PostLube_DN, ET => TF_TMR_PostLube_ET);
(* ===== CLEAR ONE-SHOT COMMANDS ===== *)
IF TRUE THEN CmdStart := FALSE; END_IF;
IF TRUE THEN CmdStop := FALSE; END_IF;
IF TRUE THEN HMI_Start := FALSE; END_IF;
IF TRUE THEN HMI_Stop := FALSE; END_IF;
IF TRUE THEN HMI_Reset := FALSE; END_IF;
END_ACTION

ACTION R05_Devices:
(* LD diagram, written out as Structured Text *)
(* ========== DEVICE CONTROL ========== *)
(* XV-101 Valve Travel Fault Detection *)
TF_TMR_XV101_IN := XV101_CmdOpen AND NOT XV101_Open OR XV101_CmdClose AND NOT XV101_Closed;
TMR_XV101(IN := TF_TMR_XV101_IN, PT := TIME#100000ms, Q => TF_TMR_XV101_DN, ET => TF_TMR_XV101_ET);
TF_TMR_XV101_Executed := TMR_XV101.ENO;
TF_Cmp_MainProgram_R05_Devices_2_1 := TF_TMR_XV101_ET > DINT_TO_TIME(CFG_ValveTimeout);
XV101_Fault := TF_Cmp_MainProgram_R05_Devices_2_1;
(* XV-102 Valve Travel Fault Detection *)
TF_TMR_XV102_IN := XV102_CmdOpen AND NOT XV102_Open OR XV102_CmdClose AND NOT XV102_Closed;
TMR_XV102(IN := TF_TMR_XV102_IN, PT := TIME#100000ms, Q => TF_TMR_XV102_DN, ET => TF_TMR_XV102_ET);
TF_TMR_XV102_Executed := TMR_XV102.ENO;
TF_Cmp_MainProgram_R05_Devices_4_1 := TF_TMR_XV102_ET > DINT_TO_TIME(CFG_ValveTimeout);
XV102_Fault := TF_Cmp_MainProgram_R05_Devices_4_1;
(* ===== COOLER FAN CONTROL ===== *)
TF_Cmp_MainProgram_R05_Devices_5_1 := TT301_PV > CFG_FanOnTemp;
IF TF_Cmp_MainProgram_R05_Devices_5_1 THEN FanCmd := TRUE; END_IF;
TF_Cmp_MainProgram_R05_Devices_6_1 := TT301_PV < CFG_FanOffTemp;
IF TF_Cmp_MainProgram_R05_Devices_6_1 THEN FanCmd := FALSE; END_IF;
(* Stop fan if not running or starting *)
IF NOT StsRunning AND NOT StsStarting THEN FanCmd := FALSE; END_IF;
END_ACTION

ACTION R06_Control:
(* LD diagram, written out as Structured Text *)
(* ========== PID DISCHARGE PRESSURE CONTROL ==========
================= SIMPLE PID SIMULATION =============== *)
(* PID Setpoint from HMI *)
PID_SP := HMI_SP_Press;
(* PID Process Value *)
PID_PV := PT102_PV;
(* PID Error Calculation *)
IF PID_Enable AND NOT PT102_Fault THEN PID_Err := PID_SP - PID_PV; END_IF;
(* PID Output = Kp*Err + Integral *)
_MUL1037_EN := PID_Enable AND PID_Auto;
IF _MUL1037_EN THEN PID_Out := PID_Kp * PID_Err; END_IF;
IF _MUL1037_EN THEN ASC_Flow := PID_Ki * PID_Err; END_IF;
IF _MUL1037_EN THEN ASC_Flow := ASC_Flow * ScanTime; END_IF;
IF _MUL1037_EN THEN PID_Int := PID_Int + ASC_Flow; END_IF;
IF _MUL1037_EN THEN PID_Out := PID_Out + PID_Int; END_IF;
(* Clamp Output High *)
TF_Cmp_MainProgram_R06_Control_5_1 := PID_Out > CFG_SpeedMax;
IF TF_Cmp_MainProgram_R06_Control_5_1 THEN PID_Out := CFG_SpeedMax; END_IF;
(* Clamp Output Low *)
TF_Cmp_MainProgram_R06_Control_6_1 := PID_Out < CFG_SpeedMin;
IF TF_Cmp_MainProgram_R06_Control_6_1 THEN PID_Out := CFG_SpeedMin; END_IF;
(* Anti-Windup: Clamp Integral *)
TF_Cmp_MainProgram_R06_Control_7_1 := PID_Int > 50.0;
IF TF_Cmp_MainProgram_R06_Control_7_1 THEN PID_Int := 50.0; END_IF;
TF_Cmp_MainProgram_R06_Control_8_1 := PID_Int < (-50.0);
IF TF_Cmp_MainProgram_R06_Control_8_1 THEN PID_Int := -50.0; END_IF;
(* ========== ANTI-SURGE CONTROL ==========
========== SIMPLE ASC SIMULATION ========= *)
ASC_Flow := FT101_PV;
(* Calculate Pressure Ratio *)
TF_Cmp_MainProgram_R06_Control_10_1 := PT101_PV > 0.1;
IF TF_Cmp_MainProgram_R06_Control_10_1 THEN ASC_PressRatio := PT102_PV / PT101_PV; END_IF;
(* Simplified Surge Limit Calculation *)
ASC_SurgeLimit := ASC_PressRatio - 1.0;
ASC_SurgeLimit := ASC_SurgeLimit * 2000.0;
ASC_SurgeLimit := ASC_SurgeLimit + 1000.0;
(* Surge Margin (%) *)
TF_Cmp_MainProgram_R06_Control_12_1 := ASC_SurgeLimit > 0.0;
IF TF_Cmp_MainProgram_R06_Control_12_1 THEN ASC_SurgeMargin := ASC_Flow - ASC_SurgeLimit; END_IF;
IF TF_Cmp_MainProgram_R06_Control_12_1 THEN ASC_SurgeMargin := ASC_SurgeMargin / ASC_SurgeLimit; END_IF;
IF TF_Cmp_MainProgram_R06_Control_12_1 THEN ASC_SurgeMargin := ASC_SurgeMargin * 100.0; END_IF;
(* Surge Index (0=safe, 100=surge) *)
ASC_SurgeIndex := 100.0 - ASC_SurgeMargin;
TF_Cmp_MainProgram_R06_Control_14_1 := ASC_SurgeIndex < 0.0;
IF TF_Cmp_MainProgram_R06_Control_14_1 THEN ASC_SurgeIndex := 0.0; END_IF;
TF_Cmp_MainProgram_R06_Control_15_1 := ASC_SurgeIndex > 100.0;
IF TF_Cmp_MainProgram_R06_Control_15_1 THEN ASC_SurgeIndex := 100.0; END_IF;
(* Low Margin Alarm *)
TF_Cmp_MainProgram_R06_Control_16_1 := ASC_SurgeMargin < CFG_SurgeMarginAlm;
ASC_LowMarginAlm := TF_Cmp_MainProgram_R06_Control_16_1;
(* Open Recycle When Margin Low *)
IF ASC_Enable AND ASC_Auto THEN TF_Cmp_MainProgram_R06_Control_17_1 := ASC_SurgeMargin < ASC_MarginSP; END_IF;
IF ASC_Enable AND ASC_Auto AND TF_Cmp_MainProgram_R06_Control_17_1 THEN ASC_RecycleCmd := ASC_RecycleCmd + 1.0; END_IF;
(* Close Recycle When Margin OK *)
IF ASC_Enable AND ASC_Auto THEN TF_Cmp_MainProgram_R06_Control_18_1 := ASC_SurgeMargin >= ASC_MarginSP; END_IF;
IF ASC_Enable AND ASC_Auto AND TF_Cmp_MainProgram_R06_Control_18_1 THEN ASC_RecycleCmd := ASC_RecycleCmd - 0.1; END_IF;
(* Minimum Recycle While Running *)
IF StsRunning THEN TF_Cmp_MainProgram_R06_Control_19_1 := ASC_RecycleCmd < CFG_RecycleMinRun; END_IF;
IF StsRunning AND TF_Cmp_MainProgram_R06_Control_19_1 THEN ASC_RecycleCmd := CFG_RecycleMinRun; END_IF;
TF_Cmp_MainProgram_R06_Control_20_1 := ASC_RecycleCmd > 100.0;
IF TF_Cmp_MainProgram_R06_Control_20_1 THEN ASC_RecycleCmd := 100.0; END_IF;
TF_Cmp_MainProgram_R06_Control_21_1 := ASC_RecycleCmd < 0.0;
IF TF_Cmp_MainProgram_R06_Control_21_1 THEN ASC_RecycleCmd := 0.0; END_IF;
(* Output to Recycle Valve *)
IF ASC_Enable THEN TF_Local_5_O_Ch0Data_4 := ASC_RecycleCmd; END_IF;
END_ACTION

ACTION R07_Alarms:
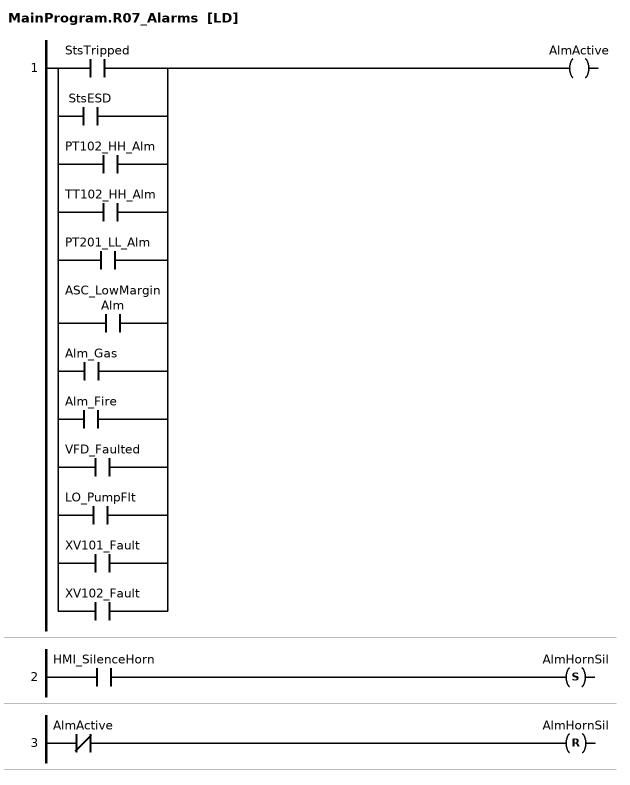
(* LD diagram, written out as Structured Text *)
(* ========== ALARM PROCESSING ========== *)
(* Combine All Alarms *)
AlmActive := StsTripped OR StsESD OR PT102_HH_Alm OR TT102_HH_Alm OR PT201_LL_Alm OR ASC_LowMarginAlm OR Alm_Gas OR Alm_Fire OR VFD_Faulted OR LO_PumpFlt OR XV101_Fault OR XV102_Fault;
(* Silence Horn Command *)
IF HMI_SilenceHorn THEN AlmHornSil := TRUE; END_IF;
(* Reset Silence When All Clear *)
IF NOT AlmActive THEN AlmHornSil := FALSE; END_IF;
END_ACTION

ACTION R08_Outputs:
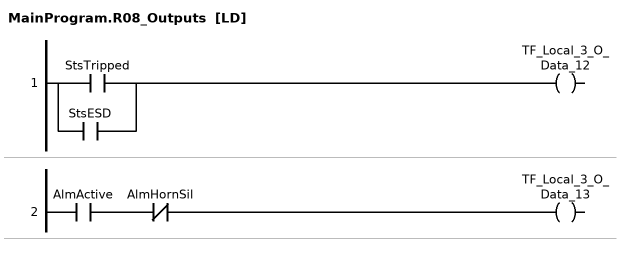
(* LD diagram, written out as Structured Text *)
TF_Local_3_O_Data_12 := StsTripped OR StsESD;
(* ===== ALARM OUTPUTS ===== *)
TF_Local_3_O_Data_13 := AlmActive AND NOT AlmHornSil;
END_ACTION
END_PROGRAM

CONFIGURATION Application
  RESOURCE Application ON PLC
    VAR_GLOBAL  (* ControllerTags *)
      AlmActive : BOOL;  (* Compressor Alarm Active *)
      AlmHornSil : BOOL := FALSE;
      Alm_Fire : BOOL;
      Alm_Gas : BOOL;
      Alm_Vib : BOOL;
      ASC_Auto : BOOL := FALSE;  (* Anti Surge Control to Aut *)
      ASC_Enable : BOOL := FALSE;  (* Anti Surge Control Enable *)
      ASC_Flow : REAL := 0.0;  (* Anti Surge Control Flow *)
      ASC_Ki : REAL := 1.0;  (* Anti Surge Control Ki *)
      ASC_Kp : REAL := 5.0;  (* Anti Surge Control Kp *)
      ASC_LowMarginAlm : BOOL := FALSE;  (* Anti Surge Control Low Margine Alarm *)
      ASC_MarginSP : REAL := 15.0;  (* Anti Surge Control Magin SP *)
      ASC_PressRatio : REAL := 0.0;  (* Anti Surge Control Pressure Ratio *)
      ASC_RecycleCmd : REAL := 0.0;  (* Anti Surge Control Recycle Cmd *)
      ASC_SurgeIndex : REAL := 0.0;  (* Anti Surge Control Surge Index *)
      ASC_SurgeLimit : REAL := 0.0;  (* Anti Surge Control Surge Limit *)
      ASC_SurgeMargin : REAL := 0.0;  (* Anti Surge Control Surge Margin *)
      BDV101_Closed : BOOL;
      BDV101_CmdOpen : BOOL;  (* Open Cmd BDV-101 Blowdown Vavle *)
      BDV101_Open : BOOL;
      CFG_FanOffTemp : REAL := 35.0;  (* Cooler Fan Off Temp (C) *)
      CFG_FanOnTemp : REAL := 45.0;  (* Cooler Fan On Temp (C) *)
      CFG_LO_Press_Min : REAL := 2.0;  (* Min Lube Oil Pressure (barg) *)
      CFG_PostLubeTime : DINT := 120000;  (* Post-Lube Time Normal (ms) *)
      CFG_PostLubeTripTime : DINT := 300000;  (* Post-Lube Time After Trip (ms) *)
      CFG_PrelubeTime : DINT := 5000;  (* Prelube Time Required (ms) *)
      CFG_PrelubeTimeout : DINT := 60000;  (* Prelube Timeout (ms) *)
      CFG_PT102_H : REAL := 100.0;  (* Discharge Press High Alarm (barg) *)
      CFG_PT102_HH : REAL := 120.0;  (* Discharge Press HH Trip (barg) *)
      CFG_PT201_L : REAL := 2.0;  (* Lube Oil Press Low Alarm (barg) *)
      CFG_PT201_LL : REAL := 1.0;  (* Lube Oil Press LL Trip (barg) *)
      CFG_RecycleMinRun : REAL := 10.0;  (* Min Recycle While Running (%) *)
      CFG_RecycleShutdown : REAL := 50.0;  (* Recycle for Shutdown (%) *)
      CFG_SpeedMax : REAL := 100.0;  (* VFD Max Speed (%) *)
      CFG_SpeedMin : REAL := 30.0;  (* VFD Min Speed (%) *)
      CFG_SpeedStart : REAL := 30.0;  (* VFD Start Speed (%) *)
      CFG_SurgeMarginAlm : REAL := 15.0;  (* Surge Margin Alarm (%) *)
      CFG_SurgeMarginTrip : REAL := 10.0;  (* Surge Margin Trip (%) *)
      CFG_TripDelay : DINT := 2000;  (* Process Trip Delay (ms) *)
      CFG_TT102_H : REAL := 160.0;  (* Discharge Temp High Alarm (C) *)
      CFG_TT102_HH : REAL := 180.0;  (* Discharge Temp HH Trip (C) *)
      CFG_ValveTimeout : DINT := 30000;  (* Valve Travel Timeout (ms) *)
      CFG_VFDStartTimeout : DINT := 10000;  (* VFD Start Timeout (ms) *)
      CFG_WarmupTime : DINT := 60000;  (* Warmup Time (ms) *)
      CmdReset : BOOL := FALSE;
      CmdStart : BOOL := FALSE;
      CmdStop : BOOL := FALSE;
      CV101_Cmd : REAL := 0.0;  (* CV-101 Recycle Valve Command (%) *)
      FanCmd : BOOL;  (* Fan Cmd (1=Start,0=Stop) *)
      FanFlt : BOOL;
      FanRun : BOOL;
      FT101_Fault : BOOL;
      FT101_PV : REAL;  (* FT-101 Compressor Flow (m3/h) *)
      HMI_Reset : BOOL := FALSE;  (* Reset Cmd from HMI *)
      HMI_SilenceHorn : BOOL := FALSE;  (* Silence Horn Cmd from HMI *)
      HMI_SP_Press : REAL := 80.0;
      HMI_Start : BOOL := FALSE;  (* Start Cmd from HMI *)
      HMI_Stop : BOOL := FALSE;  (* Stop Cmd from HMI *)
      LO_PressOK : BOOL := FALSE;  (* LO Pressure OK *)
      LO_PumpCmd : BOOL;  (* LO Pump Cmd - Start *)
      LO_PumpFlt : BOOL;
      LO_PumpRun : BOOL;
      ModeLocal : BOOL := FALSE;  (* Local Mode *)
      ModeRemote : BOOL := FALSE;  (* Remote Mode *)
      ONS_Reset : BOOL := FALSE;
      ONS_Start : BOOL := FALSE;
      ONS_Trip : BOOL := FALSE;
      PermOK : BOOL := FALSE;
      Perm_BDV : BOOL := FALSE;  (* Permissive BDV-101 Blowdown Valve *)
      Perm_ESD : BOOL;
      Perm_Instr : BOOL := FALSE;
      Perm_LO_Lvl : BOOL;
      Perm_NoTrip : BOOL := FALSE;
      Perm_VFD : BOOL := FALSE;
      PID_Auto : BOOL := FALSE;  (* PID Mode - Auto *)
      PID_Enable : BOOL := FALSE;  (* PID Enable Cmd *)
      PID_Err : REAL := 0.0;  (* PID Error *)
      PID_Int : REAL := 0.0;  (* PID Interlock *)
      PID_Ki : REAL := 0.5;  (* PID Ki *)
      PID_Kp : REAL := 2.0;  (* PID Kp *)
      PID_Out : REAL := 0.0;  (* PID CV *)
      PID_PV : REAL := 0.0;  (* PID PV *)
      PID_SP : REAL := 80.0;  (* PID Discharge Press SP (barg) *)
      PT101_Fault : BOOL;  (* PT-101 Suction Pressure Fault *)
      PT101_PV : REAL;  (* PT-101 Suction Pressure (barg) *)
      PT102_Fault : BOOL;  (* PT-102 Discharge Pressure Fault *)
      PT102_HH_Alm : BOOL := FALSE;  (* PT-102 Discharge Pressure High-High Alarm *)
      PT102_H_Alm : BOOL := FALSE;  (* PT-102 Discharge Pressure High Alarm *)
      PT102_PV : REAL;  (* PT-102 Discharge Pressure (barg) *)
      PT201_Fault : BOOL;  (* PT-201 Lube Oil Pressure Fault *)
      PT201_LL_Alm : BOOL := FALSE;  (* PT-201 Lube Oil Pressure Low-Low Alarm *)
      PT201_L_Alm : BOOL := FALSE;  (* PT-201 Lube Oil Pressure Low Alarm *)
      PT201_PV : REAL;  (* PT-201 Lube Oil Pressure (barg) *)
      RunHours : REAL := 0.0;
      ScanTime : REAL := 0.1;
      StartCount : DINT := 0;
      State : DINT := 0;  (* State: 0=Stop 10=Prelube 20=Valves 30=VFDStart 40=Warmup 50=Run 60=Stop 90=Trip 95=ESD *)
      StsESD : BOOL := FALSE;  (* ESD Status (1=ESD, 0=Healthy) *)
      StsReady : BOOL;  (* Compressor Ready *)
      StsRunning : BOOL;  (* Compressor Running *)
      StsStarting : BOOL := FALSE;  (* Compressor Starting *)
      StsStopped : BOOL := FALSE;  (* Compressor Stopped *)
      StsStopping : BOOL := FALSE;  (* Compressor Stopping *)
      StsTripped : BOOL := FALSE;  (* Compressor Tripped *)
      TMR_PostLube : Standard.TON;
      TMR_Prelube : Standard.TON;
      TMR_Trip_DischP : Standard.TON;
      TMR_Trip_DischT : Standard.TON;
      TMR_Trip_LO : Standard.TON;
      TMR_Valve : Standard.TON;
      TMR_VFDStart : Standard.TON;
      TMR_Warmup : Standard.TON;
      TMR_XV101 : Standard.TON;
      TMR_XV102 : Standard.TON;
      TripActive : BOOL := FALSE;  (* Trip Active *)
      TripCode : DINT := 0;  (* 1=ESD 2=Fire 3=Vib 4=VFD 5=LO_P 6=DischT 7=DischP 8=Surge 9=Comms *)
      TripCount : DINT := 0;
      TripLatch : BOOL := FALSE;
      Trip_Comms : BOOL := FALSE;  (* Trip VFD Communication Fault *)
      Trip_DischP : BOOL := FALSE;  (* Discharge Pressure Trip *)
      Trip_DischT : BOOL := FALSE;  (* Discharge Temperatue Trip *)
      Trip_ESD : BOOL;
      Trip_Fire : BOOL := FALSE;  (* Fire Alarm Trip *)
      Trip_LO_P : BOOL := FALSE;  (* Lube Oil Trip *)
      Trip_Surge : BOOL := FALSE;  (* Surge Trip *)
      Trip_VFD : BOOL := FALSE;  (* Trip VFD Fault *)
      Trip_Vib : BOOL;
      TT101_Fault : BOOL;  (* TT-101 Suction Temperature Fault *)
      TT101_PV : REAL;  (* TT-101 Suction Temperature (C) *)
      TT102_Fault : BOOL;  (* TT-102 Discharge Temperature Fault *)
      TT102_HH_Alm : BOOL := FALSE;  (* TT-102 Discharge Temperature HH Alarm *)
      TT102_H_Alm : BOOL := FALSE;  (* TT-102 Discharge Temperature High Alarm *)
      TT102_PV : REAL;  (* TT-102 Discharge Temperature (C) *)
      TT201_PV : REAL;  (* TT-201 Lube Oil Temperature (C) *)
      TT301_PV : REAL;  (* TT-301 Cooler Outlet Temp (C) *)
      ValvesOpen : BOOL := FALSE;  (* Both Suction Valves Open *)
      VFD_CmdReset : BOOL;  (* Cmd to VFD - Reset *)
      VFD_CmdStart : BOOL;  (* Cmd to VFD - Start *)
      VFD_CmdStop : BOOL;  (* Cmd to VFD - Stop *)
      VFD_CommFlt : BOOL;
      VFD_Faulted : BOOL;
      VFD_Ready : BOOL;
      VFD_Running : BOOL;
      VFD_SpeedCmd : REAL := 0.0;  (* VFD Speed Command (%) *)
      XV101_Closed : BOOL;
      XV101_CmdClose : BOOL;  (* Close Cmd to XV101 Suction Vavle *)
      XV101_CmdOpen : BOOL;  (* Open Cmd - XV101 Suction Vavle *)
      XV101_Fault : BOOL := FALSE;  (* Fault XV101 Suction Vavle *)
      XV101_Open : BOOL;
      XV102_Closed : BOOL;
      XV102_CmdClose : BOOL;  (* Close Cmd to XV102 Suction Vavle *)
      XV102_CmdOpen : BOOL;  (* Open Cmd to XV102 Suction Vavle *)
      XV102_Fault : BOOL := FALSE;  (* Fault XV101 Suction Vavle *)
      XV102_Open : BOOL;
      TF_Local_1_I_Data_0 : BOOL;  (* Portable surrogate for Rockwell operand Local:1:I.Data.0 *)
      TF_Local_1_I_Data_0_2 : BOOL;  (* Portable surrogate for Rockwell operand Local:1:I.Data.0 *)
      TF_Local_1_I_Data_1 : BOOL;  (* Portable surrogate for Rockwell operand Local:1:I.Data.1 *)
      TF_Local_1_I_Data_2 : BOOL;  (* Portable surrogate for Rockwell operand Local:1:I.Data.2 *)
      TF_Local_1_I_Data_3 : BOOL;  (* Portable surrogate for Rockwell operand Local:1:I.Data.3 *)
      TF_Local_5_O_Ch1Data : REAL;  (* Portable surrogate for Rockwell operand Local:5:O.Ch1Data *)
      TF_Local_5_O_Ch1Data_2 : REAL;  (* Portable surrogate for Rockwell operand Local:5:O.Ch1Data *)
      TF_Local_5_O_Ch0Data : REAL;  (* Portable surrogate for Rockwell operand Local:5:O.Ch0Data *)
      TF_Local_5_O_Ch1Data_3 : REAL;  (* Portable surrogate for Rockwell operand Local:5:O.Ch1Data *)
      TF_Local_5_O_Ch1Data_4 : REAL;  (* Portable surrogate for Rockwell operand Local:5:O.Ch1Data *)
      TF_Local_5_O_Ch1Data_5 : REAL;  (* Portable surrogate for Rockwell operand Local:5:O.Ch1Data *)
      TF_Local_5_O_Ch1Data_6 : REAL;  (* Portable surrogate for Rockwell operand Local:5:O.Ch1Data *)
      TF_Local_5_O_Ch0Data_2 : REAL;  (* Portable surrogate for Rockwell operand Local:5:O.Ch0Data *)
      TF_Local_5_O_Ch1Data_7 : REAL;  (* Portable surrogate for Rockwell operand Local:5:O.Ch1Data *)
      TF_Local_5_O_Ch1Data_8 : REAL;  (* Portable surrogate for Rockwell operand Local:5:O.Ch1Data *)
      TF_Local_5_O_Ch0Data_3 : REAL;  (* Portable surrogate for Rockwell operand Local:5:O.Ch0Data *)
      TF_Local_5_O_Ch0Data_4 : REAL;  (* Portable surrogate for Rockwell operand Local:5:O.Ch0Data *)
      TF_Local_3_O_Data_12 : BOOL;  (* Portable surrogate for Rockwell operand Local:3:O.Data.12 *)
      TF_Local_3_O_Data_13 : BOOL;  (* Portable surrogate for Rockwell operand Local:3:O.Data.13 *)
      TF_TMR_PostLube_IN : BOOL;  (* TwinForge IEC timer IN for TMR_PostLube *)
      TF_TMR_PostLube_DN : BOOL;  (* TwinForge IEC timer DN for TMR_PostLube *)
      TF_TMR_PostLube_ET : TIME;  (* TwinForge IEC timer ET for TMR_PostLube *)
      TF_TMR_PostLube_Executed : BOOL;  (* TwinForge IEC timer Executed for TMR_PostLube *)
      TF_TMR_Prelube_IN : BOOL;  (* TwinForge IEC timer IN for TMR_Prelube *)
      TF_TMR_Prelube_DN : BOOL;  (* TwinForge IEC timer DN for TMR_Prelube *)
      TF_TMR_Prelube_ET : TIME;  (* TwinForge IEC timer ET for TMR_Prelube *)
      TF_TMR_Prelube_Executed : BOOL;  (* TwinForge IEC timer Executed for TMR_Prelube *)
      TF_TMR_Trip_DischP_IN : BOOL;  (* TwinForge IEC timer IN for TMR_Trip_DischP *)
      TF_TMR_Trip_DischP_DN : BOOL;  (* TwinForge IEC timer DN for TMR_Trip_DischP *)
      TF_TMR_Trip_DischP_ET : TIME;  (* TwinForge IEC timer ET for TMR_Trip_DischP *)
      TF_TMR_Trip_DischP_Executed : BOOL;  (* TwinForge IEC timer Executed for TMR_Trip_DischP *)
      TF_TMR_Trip_DischT_IN : BOOL;  (* TwinForge IEC timer IN for TMR_Trip_DischT *)
      TF_TMR_Trip_DischT_DN : BOOL;  (* TwinForge IEC timer DN for TMR_Trip_DischT *)
      TF_TMR_Trip_DischT_ET : TIME;  (* TwinForge IEC timer ET for TMR_Trip_DischT *)
      TF_TMR_Trip_DischT_Executed : BOOL;  (* TwinForge IEC timer Executed for TMR_Trip_DischT *)
      TF_TMR_Trip_LO_IN : BOOL;  (* TwinForge IEC timer IN for TMR_Trip_LO *)
      TF_TMR_Trip_LO_DN : BOOL;  (* TwinForge IEC timer DN for TMR_Trip_LO *)
      TF_TMR_Trip_LO_ET : TIME;  (* TwinForge IEC timer ET for TMR_Trip_LO *)
      TF_TMR_Trip_LO_Executed : BOOL;  (* TwinForge IEC timer Executed for TMR_Trip_LO *)
      TF_TMR_Valve_IN : BOOL;  (* TwinForge IEC timer IN for TMR_Valve *)
      TF_TMR_Valve_DN : BOOL;  (* TwinForge IEC timer DN for TMR_Valve *)
      TF_TMR_Valve_ET : TIME;  (* TwinForge IEC timer ET for TMR_Valve *)
      TF_TMR_Valve_Executed : BOOL;  (* TwinForge IEC timer Executed for TMR_Valve *)
      TF_TMR_VFDStart_IN : BOOL;  (* TwinForge IEC timer IN for TMR_VFDStart *)
      TF_TMR_VFDStart_DN : BOOL;  (* TwinForge IEC timer DN for TMR_VFDStart *)
      TF_TMR_VFDStart_ET : TIME;  (* TwinForge IEC timer ET for TMR_VFDStart *)
      TF_TMR_VFDStart_Executed : BOOL;  (* TwinForge IEC timer Executed for TMR_VFDStart *)
      TF_TMR_Warmup_IN : BOOL;  (* TwinForge IEC timer IN for TMR_Warmup *)
      TF_TMR_Warmup_DN : BOOL;  (* TwinForge IEC timer DN for TMR_Warmup *)
      TF_TMR_Warmup_ET : TIME;  (* TwinForge IEC timer ET for TMR_Warmup *)
      TF_TMR_Warmup_Executed : BOOL;  (* TwinForge IEC timer Executed for TMR_Warmup *)
      TF_TMR_XV101_IN : BOOL;  (* TwinForge IEC timer IN for TMR_XV101 *)
      TF_TMR_XV101_DN : BOOL;  (* TwinForge IEC timer DN for TMR_XV101 *)
      TF_TMR_XV101_ET : TIME;  (* TwinForge IEC timer ET for TMR_XV101 *)
      TF_TMR_XV101_Executed : BOOL;  (* TwinForge IEC timer Executed for TMR_XV101 *)
      TF_TMR_XV102_IN : BOOL;  (* TwinForge IEC timer IN for TMR_XV102 *)
      TF_TMR_XV102_DN : BOOL;  (* TwinForge IEC timer DN for TMR_XV102 *)
      TF_TMR_XV102_ET : TIME;  (* TwinForge IEC timer ET for TMR_XV102 *)
      TF_TMR_XV102_Executed : BOOL;  (* TwinForge IEC timer Executed for TMR_XV102 *)
    END_VAR
    TASK MainTask(PRIORITY := 10);
    PROGRAM MainProgram WITH MainTask : MainProgram;
  END_RESOURCE
END_CONFIGURATION
